Staubli VAL3: main.pgx

public program main()
  local bool l_bSave
  local bool l_bOverRide
  local bool l_bOk
  local bool l_bUnreached
  local string l_sMessage
begin
      // INIT
      call onStart()
        // LOOP UNTIL nKey=255
        nIndexItem=0
  do
    call refresh()
    nKey=getKey()
    call use:listevent(nKey,nIndex,sEvent)
    nView=use:nView
    switch nKey
      case 259
        // TAB
        bLarge=!bLarge
        //  call use:setView()
      break
      case 263
        // backSpace rename
        //call onBackEvent(l_bSave)
      break
      case 32
        // space to edit Action
        //call onSpaceEvent()
      break
      case 271
        call onF1Event()
      break
      case 272
        //
        call onF2Event()
      break
      case 273
        //
        call onF3Event()
      break
      case 274
        //
        call onF4Event()
      break
      case 275
        //
        call onF5Event()
      break
      //
      case 276
        call onF6Event()
      break
      case 277
        //
        call onF7Event()
      break
      case 278
        //
        call onF8Event()
      break
      case 270
        //
        call onEnterEvent()
      break
    endSwitch
    delay(0)
  until workingMode()!=4
      if workingMode()!=4 and workingMode()!=1
      call use:timerDialog("请切换至手动模式或者远程自动模式",0)
      wait(workingMode()==4 or workingMode()==1)
      delay(0)
     endIf
   use:bUseRefresh=true
      //  // exit
     call onExit(l_bSave)
end
